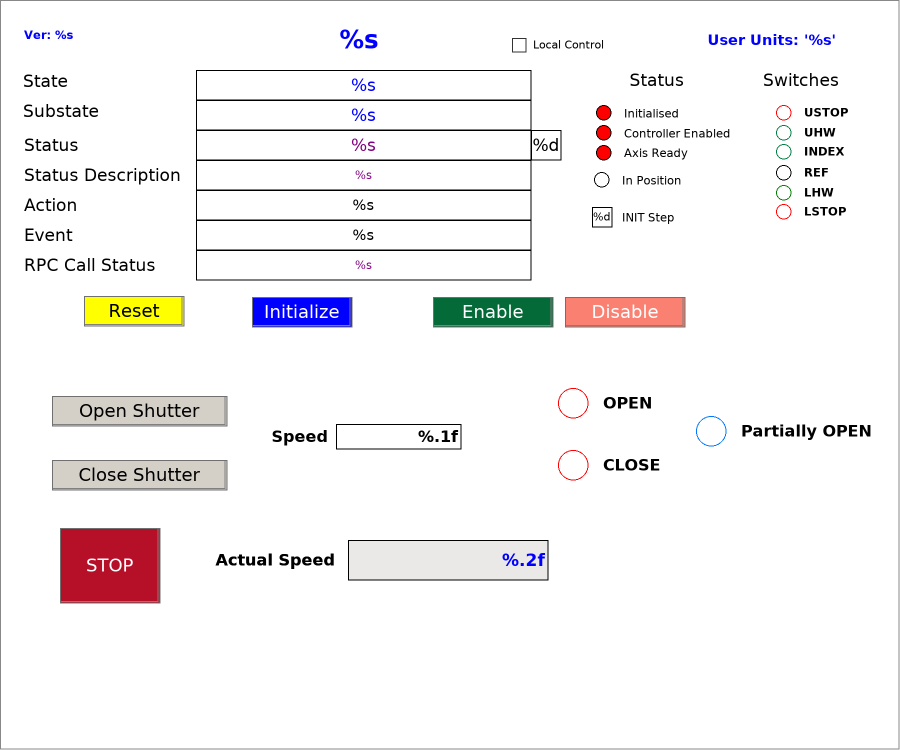
VISUALIZATION GUI_TEMPLATE_SHUTTER_CONTROL  // 900x750
VAR_IN_OUT
	m_Instance:	FB_NOTT_MOTOR;
END_VAR
VAR
	m_lrOffSet : LREAL := 0;
END_VAR
    Rectangle (196,70 335x30), "%s", text variable: m_Instance.stat.sState
    Rectangle (196,100 335x30), "%s", text variable: m_Instance.stat.sSubstate
    Button (84,296 100x30), "Reset", input disabled if: NOT m_Instance.stat.bLocal OR NOT m_Instance.in_bSafe
        OnMouseDown: execute {
            m_Instance.ctrl.bLocalCmd := TRUE;
            m_Instance.ctrl.nCommand := E_MOTOR_COMMAND.RESET;
            m_Instance.ctrl.bExecute := TRUE;
        }
    Button (252,297 100x30), "Initialize", input disabled if: NOT m_Instance.stat.bLocal OR NOT m_Instance.in_bSafe
        OnMouseDown: execute {
            m_Instance.ctrl.bLocalCmd := TRUE;
            m_Instance.ctrl.nCommand := E_MOTOR_COMMAND.INIT;
            m_Instance.ctrl.bExecute := TRUE;
        }
    Button (60,528 100x75), "STOP", input disabled if: NOT m_Instance.stat.bLocal OR NOT m_Instance.in_bSafe
        OnMouseDown: execute {
            m_Instance.ctrl.bLocalCmd := TRUE;
            m_Instance.ctrl.nCommand := E_MOTOR_COMMAND.STOP;
            m_Instance.ctrl.bExecute := TRUE;
        }
    Button (433,297 120x30), "Enable", input disabled if: NOT m_Instance.stat.bLocal OR NOT m_Instance.in_bSafe
        OnMouseDown: execute {
            m_Instance.ctrl.bLocalCmd := TRUE;
            m_Instance.ctrl.nCommand := E_MOTOR_COMMAND.ENABLE;
            m_Instance.ctrl.bExecute := TRUE;
        }
    Button (565,297 120x30), "Disable", input disabled if: NOT m_Instance.stat.bLocal OR NOT m_Instance.in_bSafe
        OnMouseDown: execute {
            m_Instance.ctrl.bLocalCmd := TRUE;
            m_Instance.ctrl.nCommand := E_MOTOR_COMMAND.DISABLE;
            m_Instance.ctrl.bExecute := TRUE;
        }
    Rectangle (20,66 170x30), "State"
    Rectangle (20,96 170x30), "Substate"
    Rectangle (196,130 335x30), "%s", text variable: m_Instance.stat.sStatus
    Rectangle (196,160 335x30), "%s", tooltip "Additional information mostly used for description of errors", text variable: m_Instance.stat.sErrorText
    Rectangle (21,130 170x30), "Status"
    Rectangle (21,160 170x30), "Status Description"
    Rectangle (196,190 335x30), "%s", text variable: m_Instance.stat.sActionDesc
    Rectangle (196,220 335x30), "%s", text variable: m_Instance.stat.sEventDesc
    Rectangle (21,190 170x30), "Action"
    Rectangle (21,220 170x30), "Event"
    Rectangle (243,22 232x35), "%s", text variable: m_Instance.sName
    Checkbox (510,30 116x30), "Local Control", variable: m_Instance.stat.bLocal
    Rectangle (611,65 92x30), "Status"
    Rectangle (531,130 30x30), "%d", text variable: m_Instance.stat.nStatus
    Rectangle (755,65 92x30), "Switches"
    Rectangle (801,105 50x15), "USTOP"
    Ellipse (776,105 15x15), colour toggle: m_Instance.stat.signals[5].bActive
    Ellipse (776,125 15x15), colour toggle: m_Instance.stat.signals[4].bActive
    Ellipse (776,185 15x15), colour toggle: m_Instance.stat.signals[1].bActive
    Ellipse (776,204 15x15), colour toggle: m_Instance.stat.signals[0].bActive
    Ellipse (776,165 15x15), colour toggle: m_Instance.stat.signals[2].bActive
    Rectangle (801,144 50x15), "INDEX"
    Rectangle (801,125 50x15), "UHW"
    Rectangle (801,165 50x15), "REF"
    Rectangle (801,185 50x15), "LHW"
    Rectangle (801,204 50x15), "LSTOP"
    Ellipse (776,144 15x15), colour toggle: m_Instance.stat.signals[3].bActive
    Ellipse (596,105 15x15), tooltip "GREEN = Initialised RED = Not Initialised", text variable: m_Instance.stat.bInitialised, colour toggle: m_Instance.stat.bInitialised
    Rectangle (621,101 90x25), "Initialised"
    Rectangle (621,121 125x25), "Controller Enabled"
    Rectangle (621,141 90x24), "Axis Ready"
    Ellipse (596,125 15x15), tooltip "GREEN = Enabled RED = Disabled", colour toggle: m_Instance.stat.bEnabled
    Ellipse (596,145 15x15), tooltip "GREEN = Ready RED = Not Ready", colour toggle: m_Instance.stat.bAxisReady
    Rectangle (592,207 20x20), "%d", text variable: m_Instance.stat.nInitStep
    Rectangle (619,205 90x25), "INIT Step"
    Rectangle (21,250 170x30), "RPC Call Status"
    Rectangle (196,250 335x30), "%s", text variable: m_Instance.stat.sRPCErrorText
    Rectangle (619,168 90x25), "In Position"
    Ellipse (594,172 15x15), tooltip "GREEN = In Position BLANK = Not In Position (or not used)", colour toggle: (m_Instance.stat.bInPosition) <> 0
    Rectangle (636,25 203x30), "User Units: '%s'", text variable: m_Instance.stat.axis.sUnits
    Rectangle (21,20 99x30), "Ver: %s", tooltip "'Motor.library version'", text variable: m_Instance.stat.sLibVersion, input disabled if: true
    Group (188,540 360x40)
        Rectangle (160,0 200x40), "%.2f", text variable: m_Instance.stat.lrVelActual, input disabled if: false
        Rectangle (0,5 150x30), "Actual Speed"
    Rectangle (348,540 200x40), "%.2f", text variable: m_Instance.stat.lrVelActual, input disabled if: false
    Rectangle (188,545 150x30), "Actual Speed"
    Rectangle (236,424 95x25), "Speed", tooltip "Shutter Speed (mm/sec)"
    Rectangle (336,424 125x25), "%.1f", text variable: m_Instance.ctrl.lrVelocity
        OnMouseDown: write the text variable via Default
    Button (52,396 175x30), "Open Shutter", input disabled if: NOT m_Instance.stat.bLocal OR NOT m_Instance.in_bSafe
        OnMouseDown: execute {
            m_Instance.ctrl.bLocalCmd := TRUE;
            m_Instance.ctrl.nCommand := E_MOTOR_COMMAND.MOTOR_MOVE;
            m_Instance.ctrl.nMoveType := E_MOTOR_MOVE_TYPE.VELOCITY;
            m_Instance.ctrl.nDirection := MC_Negative_Direction;
            m_Instance.ctrl.bExecute := TRUE;
        }
    Button (52,460 175x30), "Close Shutter", input disabled if: NOT m_Instance.stat.bLocal OR NOT m_Instance.in_bSafe
        OnMouseDown: execute {
            m_Instance.ctrl.bLocalCmd := TRUE;
            m_Instance.ctrl.nCommand := E_MOTOR_COMMAND.MOTOR_MOVE;
            m_Instance.ctrl.nMoveType := E_MOTOR_MOVE_TYPE.VELOCITY;
            m_Instance.ctrl.nDirection := MC_Positive_Direction;
            m_Instance.ctrl.bExecute := TRUE;
        }
    Ellipse (558,388 30x30), colour toggle: m_Instance.stat.signals[0].bActive
    Rectangle (600,388 100x30), "OPEN", tooltip "Shutter is Open"
    Ellipse (558,450 30x30), colour toggle: m_Instance.stat.signals[5].bActive
    Rectangle (600,450 100x30), "CLOSE", tooltip "Shutter is closed"
    Ellipse (696,416 30x30), colour toggle: m_Instance.bShutterPartiallyOpen
    Rectangle (738,416 143x30), "Partially OPEN", tooltip "Either shutter is opening or closing"
END_VISUALIZATION

(* stored: Version 1.1.0.1, ProductVersion 3.1.4024.14
   Visu GUI_TEMPLATE_SHUTTER_CONTROL: Id {1767135e-a2fe-4351-a2a4-0c445864d466} *)
